FUNCTION_BLOCK ConditionSWITCH_CASE (* Test FB fpr Switch Statement *)
  (* Standard: 61499-2; Description: It checks if the input data I is: = 5 = 10 Copyright (c) 2019 Jan Holzweber This program and the accompanying materials are made available under the terms of the Eclipse Public License 2.0 which is available at https://www.eclipse.org/legal/epl-2.0/ SPDX-License-Identifier: EPL-2.0 *)
  (* Version 1.0, 2019-06-05, jholz *)
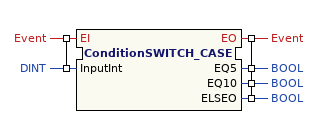
  EVENT_INPUT
    EI WITH InputInt;
  END_EVENT
  EVENT_OUTPUT
    EO WITH EQ5, EQ10, ELSEO;
  END_EVENT
  VAR_INPUT
    InputInt : DINT;
  END_VAR
  VAR_OUTPUT
    EQ5 : BOOL;
    EQ10 : BOOL;
    ELSEO : BOOL;
  END_VAR
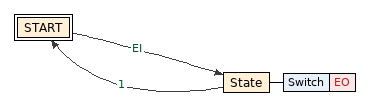
  EC_STATES
    START; (* Initial State *)
    State : Switch -> EO;
  END_STATES
  EC_TRANSITIONS
    START TO State := EI;
    State TO START := 1;
  END_TRANSITIONS
  ALGORITHM Switch IN ST:
CASE InputInt OF
	5 : EQ5 := true;
	10: EQ10 :=true;
ELSE
	ELSEO:=true;
END_CASE;
  END_ALGORITHM
END_FUNCTION_BLOCK
